// TIA Portal V20 export
DATA_BLOCK "DriveDiagConfig"   // DB18
TITLE = DriveDiagConfig
AUTHOR : Siemens Digital Industries
FAMILY : LAF
NAME : LAF_DriveDiagConfigData
VERSION : 1.1
// Configuration data array for drive diagnostic
// stored: MemoryReserve 100
   VAR
      driveObjects : Array[0..41] of "LAF_typeDriveDiagConfig";
   END_VAR
BEGIN
   driveObjects[0].referenceDesignator := WSTRING#'BA030AZSDR1';
   driveObjects[1].referenceDesignator := WSTRING#'BA030AZSDR2';
   driveObjects[2].referenceDesignator := WSTRING#'BA030AZSDR3';
   driveObjects[3].referenceDesignator := WSTRING#'';
   driveObjects[4].referenceDesignator := WSTRING#'BA030AZSDR5';
   driveObjects[5].referenceDesignator := WSTRING#'BA030AZSDR6';
   driveObjects[6].referenceDesignator := WSTRING#'BA030AZSDR7';
   driveObjects[7].referenceDesignator := WSTRING#'BA030AZSDR8';
   driveObjects[8].referenceDesignator := WSTRING#'BA030AZSDR9';
   driveObjects[9].referenceDesignator := WSTRING#'BA030AZSDR10';
   driveObjects[10].referenceDesignator := WSTRING#'BA030AZSDR11';
   driveObjects[11].referenceDesignator := WSTRING#'BA030AZSDR12';
   driveObjects[12].referenceDesignator := WSTRING#'BA030AZSDR13';
   driveObjects[13].referenceDesignator := WSTRING#'BA030AZSDR14';
   driveObjects[14].referenceDesignator := WSTRING#'BA030AZSDR15';
   driveObjects[15].referenceDesignator := WSTRING#'BA030AZSDR16';
   driveObjects[16].referenceDesignator := WSTRING#'BA030AZSDR17';
   driveObjects[17].referenceDesignator := WSTRING#'BA030AZSDR18';
   driveObjects[18].referenceDesignator := WSTRING#'BA030AZSDR19';
   driveObjects[19].referenceDesignator := WSTRING#'BA030AZSDR20';
   driveObjects[20].referenceDesignator := WSTRING#'BA030AZSDR21';
   driveObjects[21].referenceDesignator := WSTRING#'BA030AZSDR22';
   driveObjects[22].referenceDesignator := WSTRING#'BA030AZSDR23';
   driveObjects[23].referenceDesignator := WSTRING#'BA030AZSDR24';
   driveObjects[24].referenceDesignator := WSTRING#'BA030AZSDR25';
   driveObjects[25].referenceDesignator := WSTRING#'BA030AZSDR26';
   driveObjects[26].referenceDesignator := WSTRING#'BA030AZSDR27';
   driveObjects[27].referenceDesignator := WSTRING#'BA030AZSDR28';
   driveObjects[28].referenceDesignator := WSTRING#'BA030AZSDR29';
   driveObjects[29].referenceDesignator := WSTRING#'BA030AZSDR30';
   driveObjects[30].referenceDesignator := WSTRING#'BA030AZSDR31';
   driveObjects[31].referenceDesignator := WSTRING#'BA030AZSDR32';
   driveObjects[32].referenceDesignator := WSTRING#'BA030AZSDR33';
   driveObjects[33].referenceDesignator := WSTRING#'BA030AZSDR34';
   driveObjects[34].referenceDesignator := WSTRING#'BA030AZSDR35';
   driveObjects[35].referenceDesignator := WSTRING#'BA030AZSDR36';
   driveObjects[36].referenceDesignator := WSTRING#'BA030AZSDR37';
   driveObjects[37].referenceDesignator := WSTRING#'BA030AZSDR38';
   driveObjects[38].referenceDesignator := WSTRING#'BA030AZSDR39';
   driveObjects[39].referenceDesignator := WSTRING#'BA030AZSDR40';
   driveObjects[40].referenceDesignator := WSTRING#'BA030AZSDR41';
   driveObjects[41].referenceDesignator := WSTRING#'';
   driveObjects[0].axisDB := 263;
   driveObjects[1].axisDB := 141;
   driveObjects[2].axisDB := 143;
   driveObjects[3].axisDB := 0;
   driveObjects[4].axisDB := 144;
   driveObjects[5].axisDB := 145;
   driveObjects[6].axisDB := 146;
   driveObjects[7].axisDB := 147;
   driveObjects[8].axisDB := 152;
   driveObjects[9].axisDB := 151;
   driveObjects[10].axisDB := 148;
   driveObjects[11].axisDB := 149;
   driveObjects[12].axisDB := 153;
   driveObjects[13].axisDB := 150;
   driveObjects[14].axisDB := 154;
   driveObjects[15].axisDB := 155;
   driveObjects[16].axisDB := 156;
   driveObjects[17].axisDB := 157;
   driveObjects[18].axisDB := 158;
   driveObjects[19].axisDB := 159;
   driveObjects[20].axisDB := 171;
   driveObjects[21].axisDB := 172;
   driveObjects[22].axisDB := 163;
   driveObjects[23].axisDB := 162;
   driveObjects[24].axisDB := 167;
   driveObjects[25].axisDB := 166;
   driveObjects[26].axisDB := 161;
   driveObjects[27].axisDB := 160;
   driveObjects[28].axisDB := 165;
   driveObjects[29].axisDB := 164;
   driveObjects[30].axisDB := 168;
   driveObjects[31].axisDB := 169;
   driveObjects[32].axisDB := 170;
   driveObjects[33].axisDB := 177;
   driveObjects[34].axisDB := 175;
   driveObjects[35].axisDB := 178;
   driveObjects[36].axisDB := 173;
   driveObjects[37].axisDB := 174;
   driveObjects[38].axisDB := 180;
   driveObjects[39].axisDB := 179;
   driveObjects[40].axisDB := 176;
   driveObjects[41].axisDB := 0;
   driveObjects[0..2].sinaType := 124;
   driveObjects[3].sinaType := 0;
   driveObjects[4..40].sinaType := 124;
   driveObjects[41].sinaType := 0;
   driveObjects[0].sinaHwID := 259;
   driveObjects[1].sinaHwID := 517;
   driveObjects[2].sinaHwID := 818;
   driveObjects[3].sinaHwID := 0;
   driveObjects[4].sinaHwID := 519;
   driveObjects[5].sinaHwID := 523;
   driveObjects[6].sinaHwID := 527;
   driveObjects[7].sinaHwID := 529;
   driveObjects[8].sinaHwID := 541;
   driveObjects[9].sinaHwID := 547;
   driveObjects[10].sinaHwID := 559;
   driveObjects[11].sinaHwID := 561;
   driveObjects[12].sinaHwID := 564;
   driveObjects[13].sinaHwID := 569;
   driveObjects[14].sinaHwID := 568;
   driveObjects[15].sinaHwID := 571;
   driveObjects[16].sinaHwID := 573;
   driveObjects[17].sinaHwID := 577;
   driveObjects[18].sinaHwID := 659;
   driveObjects[19].sinaHwID := 660;
   driveObjects[20].sinaHwID := 589;
   driveObjects[21].sinaHwID := 596;
   driveObjects[22].sinaHwID := 654;
   driveObjects[23].sinaHwID := 667;
   driveObjects[24].sinaHwID := 671;
   driveObjects[25].sinaHwID := 682;
   driveObjects[26].sinaHwID := 620;
   driveObjects[27].sinaHwID := 626;
   driveObjects[28].sinaHwID := 684;
   driveObjects[29].sinaHwID := 686;
   driveObjects[30].sinaHwID := 605;
   driveObjects[31].sinaHwID := 635;
   driveObjects[32].sinaHwID := 663;
   driveObjects[33].sinaHwID := 690;
   driveObjects[34].sinaHwID := 649;
   driveObjects[35].sinaHwID := 692;
   driveObjects[36].sinaHwID := 657;
   driveObjects[37].sinaHwID := 697;
   driveObjects[38].sinaHwID := 665;
   driveObjects[39].sinaHwID := 666;
   driveObjects[40].sinaHwID := 653;
   driveObjects[41].sinaHwID := 0;
   driveObjects[0..1].sinaDriveObjectNo := 3;
   driveObjects[2].sinaDriveObjectNo := 4;
   driveObjects[3].sinaDriveObjectNo := 1;
   driveObjects[4].sinaDriveObjectNo := 2;
   driveObjects[5].sinaDriveObjectNo := 3;
   driveObjects[6].sinaDriveObjectNo := 4;
   driveObjects[7].sinaDriveObjectNo := 10;
   driveObjects[8].sinaDriveObjectNo := 5;
   driveObjects[9..10].sinaDriveObjectNo := 6;
   driveObjects[11].sinaDriveObjectNo := 2;
   driveObjects[12].sinaDriveObjectNo := 3;
   driveObjects[13].sinaDriveObjectNo := 4;
   driveObjects[14..40].sinaDriveObjectNo := 5;
   driveObjects[41].sinaDriveObjectNo := 1;
END_DATA_BLOCK
